FUNCTION_BLOCK IdentifyPart
VAR_INPUT
	mxEnable: BOOL;
END_VAR
VAR_OUTPUT
	Product:STRING;
	Color: STRING;
	Component: STRING;
END_VAR
VAR
	SensorReader:BYTE;
END_VAR

IF mxEnable THEN
	SensorReader.1:=gvl.ixInductiveSensor1;
	SensorReader.2:=gvl.ixInductiveSensor2;
	SensorReader.3:=gvl.ixInductiveSensor3;
	SensorReader.4:=gvl.ixInductiveSensor4;
END_IF

IF SensorReader = 0 OR SensorReader = 4 OR SensorReader = 2 OR SensorReader = 6 THEN
 	Product:='InvalidPart';
	Color := '';
	Component := 'invalidpart';
END_IF

IF SensorReader=16 THEN
	Product:='CONTAINER';
	Color := 'BLUE';
	Component := 'BLUECONTAINER';
END_IF

IF SensorReader=8 THEN
	Product:='CONTAINER';
	Color := 'YELLOW';
	Component := 'YELLOWCONTAINER';
END_IF

IF SensorReader=24 THEN
	Product:='CONTAINER';
	Color := 'RED';
	Component := 'REDCONTAINER';
END_IF

IF SensorReader=20 THEN
	Product:='CYLINDER';
	Color := 'BLUE';
	Component := 'BLUECYLINDER';
END_IF

IF SensorReader=12 THEN
	Product:='OCTAGON';
	Color := 'BLUE';
	Component := 'BLUEOCTAGON';
END_IF

IF SensorReader=28 THEN
	Product:='PLATE';
	Color := 'BLUE';
	Component := 'BLUEPLATE';
END_IF

IF SensorReader=18 THEN
	Product:='CYLINDER';
	Color := 'YELLOW';
	Component := 'YELLOWCYLINDER';
END_IF

IF SensorReader=10 THEN
	Product:='OCTAGON';
	Color := 'YELLOW';
	Component := 'YELLOWOCTAGON';
END_IF

IF SensorReader=26 THEN
	Product:='PLATE';
	Color := 'YELLOW';
	Component := 'YELLOWPLATE';
END_IF

IF SensorReader=22 THEN
	Product:='CYLINDER';
	Color := 'RED';
	Component := 'REDCYLINDER';
END_IF

IF SensorReader=14 THEN
	Product:='OCTAGON';
	Color := 'RED';
	Component := 'REDOCTAGON';
END_IF

IF SensorReader=30 THEN
	Product:='PLATE';
	Color := 'RED';
	Component := 'REDPLATE';
END_IF

END_FUNCTION_BLOCK

(* stored: Version 1.1.0.1, ProductVersion 3.1.4024.12
   POU IdentifyPart: Id {6e8fb2dd-c5ff-4951-b8f2-8618e7b10258}, SpecialFunc None *)
